FUNCTION_BLOCK FB_ChirpGen
VAR_INPUT
	EN :BOOL;
	Offset: LREAL; // where to center the chirp wave in the stroke
	StartVel :LREAL;
	EndVel :LREAL;
	A :LREAL;
	M :LREAL;
	fTIME :LREAL;
	
END_VAR
VAR_OUTPUT
	SignalOut :LREAL;
END_VAR
VAR

	RESULT: LREAL;
END_VAR

Result := A * COS (startvel * ftime + (endvel - startvel) * ftime * ftime / (2*M));
signalout := result;

END_FUNCTION_BLOCK

(* stored: Version 1.1.0.1, ProductVersion 3.1.4024.2
   POU FB_ChirpGen: Id {e265f706-1b92-434d-9e9c-2ed2746cb55a}, SpecialFunc None *)
